KUKA KRL data list: mathlib.dat

&ACCESS RV
&PARAM EDITMASK = *
&PARAM TEMPLATE = C:\KRC\Roboter\Template\vorgabe
DEFDAT mathlib PUBLIC
   ; Author:      Davide Rosa
   ; e-mail:      dddomodossola@gmail.com
   ; repository:  https://github.com/skilledAutomation/kuka_krl_wonderlibrary

   ; DESCRIPTION:
   ; This library provides a set of functions for math operations
ENDDAT
